// TIA Portal V17 export
// export: Created 2025-04-11T04:54:23.1848193Z, ExportSetting WithDefaults, DisplayName Totally Integrated Automation Portal, DisplayVersion V17, DisplayName TIA Portal Openness, DisplayVersion V17, DisplayName TIA Portal Version Control Interface, DisplayVersion V17, DisplayName SINAMICS Startdrive Advanced, DisplayVersion V17, DisplayName SINAMICS Startdrive G130, G150, S120, S150, SINAMICS MV, S210, DisplayVersion V17, DisplayName SINAMICS Startdrive G110M, G120, G120C, G120D, G120P, G115D, DisplayVersion V17, DisplayName STEP 7 Professional, DisplayVersion V17, DisplayName STEP 7 Safety, DisplayVersion V17, DisplayName WinCC Advanced, DisplayVersion V17
TYPE "UDT_EnergyData"
// stored: IsFailsafeCompliant false
   STRUCT
      rCurrentValue : Real;   // 当前能耗值
      rHourlyValue : Real;   // 小时累计值
      rDailyValue : Real;   // 日累计值
      rMonthlyValue : Real;   // 月累计值
      rYearlyValue : Real;   // 年累计值 历史数据
      aHourlyHistory : Array[0..23] of Real;   // 24小时历史数据
      aDailyHistory : Array[1..31] of Real;   // 月度每天历史数据
      aMonthlyHistory : Array[1..12] of Real;   // 年度每月历史数据 时间戳
      dtLastHourReset : DTL;   // 上次小时重置时间
      dtLastDayReset : DTL;   // 上次日重置时间
      dtLastMonthReset : DTL;   // 上次月重置时间 状态信息
      xDataValid : Bool;   // 数据有效性标志
      xError : Bool;   // 错误状态
      wStatus : Word;   // 状态字
   END_STRUCT;
END_TYPE
